{attribute 'GeneratedUsingTerminal: EK1122-0000-0018'}
{attribute addProperty BoxType "EK1122-0000-0018"}
{attribute addProperty Id "Beckhoff_EL69xxsub_EK1100EK1100_AB5A94672"}
{attribute addProperty CRC "1067022044"}
{attribute addProperty Size "2"}
TYPE Beckhoff_EL69xxEK1122_3F9976DC EXTENDS EK1122_AB5A9467 :
STRUCT
	{attribute addProperty Name "Beckhoff_EL69xxsub_EK1100"}
	Beckhoff_EL69xxsub_EK1100 : EK1100_AB5A9467;
END_STRUCT
END_TYPE

(* stored: Version 1.2.0.0, ProductVersion 3.1.4024.9
   DUT Beckhoff_EL69xxEK1122_3F9976DC: Id {ce62b6b7-5eb9-467f-839a-c02ec4b55f9a} *)
